TYPE ST_Joysticks :
STRUCT
	Left: ST_Joystick;
	Right: ST_Joystick;
END_STRUCT
END_TYPE

(* stored: Version 1.1.0.1
   DUT ST_Joysticks: Id {185991db-bd55-406a-a1ea-3602fc50608b} *)
